(* PLC project model, Beckhoff Automation Beckhoff MLlib 3.1.251201.0 *)
(* stored: creationDateTime 2026-08-04T11:42:31.0258262, modificationDateTime 2026-08-04T11:42:31.0258262 *)

TYPE ST_modelInput :
STRUCT

	{attribute 'hide'} _header_DO_NOT_CHANGE : ARRAY[0..63] OF SINT := [-1,-112,120,86,52,18,-1,-1,1,-1,0,0,-1,-1,-112,-112,-43,-24,1,0,70,-3,-76,-48,83,-35,38,69,46,-113,-109,-8,79,-112,-48,68,-59,72,65,40,-123,60,44,-49,-100,114,-78,-40,84,64,0,0,0,0,0,0,0,0,0,0,0,0,0,0];
	in_condition : ARRAY[0..0,0..3] OF REAL;
	in_direction_flag : ARRAY[0..0,0..0] OF REAL;
	in_h08_prediction_curve : ARRAY[0..0,0..2047] OF REAL;
	in_k01_prediction_curve : ARRAY[0..0,0..2047] OF REAL;

END_STRUCT
END_TYPE

TYPE ST_modelOutput :
STRUCT

	{attribute 'hide'} _header_DO_NOT_CHANGE : ARRAY[0..63] OF SINT := [-1,-112,120,86,52,18,-1,-1,1,-1,0,0,-1,-1,-112,-112,47,-22,55,-42,-127,127,-76,-92,-57,-101,61,0,2,25,93,-95,-118,113,55,-66,124,-86,30,100,58,100,45,109,73,-122,-9,80,80,-128,0,0,0,0,0,0,0,0,0,0,0,0,0,0];
	out_forward_gate : ARRAY[0..0,0..0] OF REAL;
	out_h08_centered_difference : ARRAY[0..0,0..2047] OF REAL;
	out_h08_centered_residual : ARRAY[0..0,0..2047] OF REAL;
	out_h08_mean : ARRAY[0..0,0..0] OF REAL;
	out_k01_centered_curve : ARRAY[0..0,0..2047] OF REAL;
	out_k01_mean : ARRAY[0..0,0..0] OF REAL;
	out_learned_h08_gate : ARRAY[0..0,0..0] OF REAL;
	out_prediction_curve : ARRAY[0..0,0..2047] OF REAL;

END_STRUCT
END_TYPE
